// A body that never finishes must be stopped by the deadline rather than stalling
// the suite. Tick both detects the expiry and records it - the runner only has to
// notice it happened.
//
// Called AFTER the body has run, so a budget of one allows one execution.
FUNCTION_BLOCK TEST_JournalTimesOutOnCycles IMPLEMENTS I_Test
VAR
	Subject : TestJournal;
	Budgets : ST_TestBudgets;

	Expired		 : BOOL;
	ExpectedKind : E_FailureKind;
	ActualKind	 : E_FailureKind;
	ExpectedStatus : E_TestStatus;
	ActualStatus   : E_TestStatus;
END_VAR

METHOD Run : BOOL
VAR_INPUT
	Enable : BOOL;
	Test   : I_TestAssertions;
END_VAR
Budgets.Body.Cycles	     := 2;
Budgets.Body.IsCyclesSet := TRUE;
Subject.SetBudgets(Budgets);

Subject.Begin('slow', '');

Expired := Subject.Tick();
Test.AssertFalse(Expired, 'a budget of two survives one scan');

Expired := Subject.Tick();
Test.AssertTrue(Expired, 'and expires on the second');

ExpectedKind := E_FailureKind.Timeout;
ActualKind	 := Subject.Kind;
Test.AssertEqual(ExpectedKind, ActualKind, 'recorded as a timeout');

// Tick finishes the journal itself; the runner does not have to.
ExpectedStatus := E_TestStatus.Failed;
ActualStatus   := Subject.Status;
Test.AssertEqual(ExpectedStatus, ActualStatus, 'terminal without further help');

Expired := Subject.Tick();
Test.AssertFalse(Expired, 'and does not fire twice');

Run := TRUE;
END_METHOD

END_FUNCTION_BLOCK

(* stored: Version 1.1.0.1, ProductVersion 3.1.4026.18
   POU TEST_JournalTimesOutOnCycles: Id {db17921c-2d1a-45e1-9433-45d1a6d0985c}, SpecialFunc None
   Folder I_Test: Id {d179d7ec-ff48-4c63-acb7-924e80baba8b}
   Method Run: Id {8bbed274-bc97-423f-a1c1-1e094d8de662} *)
